FUNCTION_BLOCK FB_CHPSystem EXTENDS FB_SystemContinous
VAR_INPUT
	aHeatCounterTelegramm : ARRAY[1..cMBUS_MaxTelegrams] OF ST_MBus_Data2;
END_VAR
VAR_OUTPUT
	bSetStatusOnFeedback : BOOL; //Feedback if CHP unit should be switched on to be sent to supply air valve
END_VAR
VAR	
	//chp
	CHP : FB_CHP;

	//pump
	stPU32xDefaultParameters : ST_PumpGrundfosMagna3DefaultParameters;
	PU32x : FB_PumpGrundfosMagna3 := (ST_DefaultParameters := stPU32xDefaultParameters);
	
	//valves
	stSV32xDefaultParameters : ST_DiscreteValveDefaultParameters := (nFeedback := 3);
	stRV32xDefaultParameters : ST_MixingValveDefaultParameters := (bFeedbackSignal := TRUE, tTaskCycleTime := GlobalVariables.tTaskCycleTime_MAIN, tCtrlCycleTime := GlobalVariables.tCtrlCycleTime_MAIN);	
	SV32x : FB_DiscreteValve := (ST_DefaultParameters := stSV32xDefaultParameters);
	RV32x : FB_MixingValve := (ST_DefaultParameters := stRV32xDefaultParameters);
	WMZ32x : FB_MollineC3HeatCounter();
	
	//internal variables
	bSetStatusOn_CHP   : BOOL;
	bSetStatusOn_PU32x : BOOL;
	bSetStatusOn_SV32x : BOOL;
	bSetStatusOn_RV32x : BOOL; 	
	
	//timer
	bStartTimer : BOOL;
	Timer : TON;
END_VAR

bSetStatusOnFeedback := bSetStatusOn;

//use timer because valve has no feedback signal (75 sec)
Timer(IN := bStartTimer,
	PT := T#75S);

MAIN();
CHP.GetState();
CHP(fSetPointAutomatic := 100,
	bSetStatusOnAutomatic := bSetStatusOn_CHP,
	bAlgorithmPermission := bAlgorithmPermission,
	nControlModeAutomatic := 0,
	fExternalFeedTemperature := PU32x.fTemperatureInternal);
CHP.SetState();

SV32x.GetState_BI();
SV32x(bSetStatusOnAutomatic := bSetStatusOn_SV32x,
	bAlgorithmPermission := bAlgorithmPermission);
SV32x.SetState_BO();

RV32x.GetState_AI();
RV32x(fSetPointAutomatic := fSetPoint,
	bSetStatusOnAutomatic := bSetStatusOn_RV32x,
	bAlgorithmPermission := bAlgorithmPermission,
	fTemperatureExternal := PU32x.fTemperatureInternal,
	nControlModeAutomatic := 2);
RV32x.SetState_AO();

PU32x.GetState_Profibus();
PU32x(fSetPointAutomatic := 100,
	bSetStatusOnAutomatic := bSetStatusOn_PU32x,
	bAlgorithmPermission := bAlgorithmPermission,
	nControlModeAutomatic := 0);
PU32x.SetState_Profibus();

WMZ32x(aHeatCounterTelegramm := aHeatCounterTelegramm);

METHOD PROTECTED  CheckError : BOOL
VAR_INPUT
END_VAR
VAR
	bError_PU32x : BOOL;
	//bError_CHP : BOOL;
END_VAR
VAR_OUTPUT
	bError : BOOL;
END_VAR
//check pumps for errors
bError_PU32x := PU32x.bError;
//bError_CHP := CHP.bError;

//bError := bError_PU32x OR bError_CHP;
bError := bError_PU32x;
END_METHOD

METHOD PROTECTED  Operational : BOOL
VAR_INPUT
END_VAR
VAR_OUTPUT
	bSwitchToWorking : BOOL := FALSE;
END_VAR
bSetStatusOn_CHP := TRUE;

//IF CHP.bStatusOn THEN
bStartTimer := TRUE;
IF TIMER.Q THEN
	bSwitchToWorking := TRUE;
	bStartTimer := FALSE;
END_IF
END_METHOD

METHOD PROTECTED  RampDown : BOOL
VAR_INPUT
END_VAR
VAR_OUTPUT
	bRampDownFinished : BOOL := FALSE;
END_VAR
bSetStatusOn_CHP := FALSE;

//IF NOT CHP.bStatusOn THEN
bStartTimer := TRUE;
IF Timer.Q THEN
	bSetStatusOn_PU32x := FALSE;
	bStartTimer := FALSE;
END_IF

IF NOT PU32x.bStatusOn THEN
	bSetStatusOn_RV32x := FALSE;
	bSetStatusOn_SV32x := FALSE;

	IF SV32x.bStatusOn THEN
		bRampDownFinished := TRUE;
	END_IF
END_IF
END_METHOD

METHOD PROTECTED  RampUp : BOOL
VAR_INPUT
END_VAR
VAR_OUTPUT
	bRampUpFinished : BOOL := FALSE;
END_VAR
bSetStatusOn_SV32x := TRUE;
bSetStatusOn_RV32x := TRUE;

IF SV32x.bStatusOn THEN
	bSetStatusOn_PU32x := TRUE;
END_IF

IF PU32x.bStatusOn THEN
	bStartTimer := FALSE; //resets timer	
	bRampUpFinished := TRUE;
END_IF
END_METHOD

METHOD PROTECTED   SetSetPointLimits : BOOL
VAR_INPUT
END_VAR
aSetPointLimits[1] := CHP.ST_DefaultParameters.aSetPointLimitsTemperature[1];
aSetPointLimits[2] := CHP.ST_DefaultParameters.aSetPointLimitsTemperature[2];
END_METHOD

METHOD PROTECTED  Working : BOOL
VAR_INPUT
END_VAR
VAR_OUTPUT
	bSwitchToOperational : BOOL := FALSE;
END_VAR
//empty method
END_METHOD

END_FUNCTION_BLOCK

(* stored: Version 1.1.0.1, ProductVersion 3.1.4024.10
   POU FB_CHPSystem: Id {03be9f87-4e59-4877-a478-dceefb67f1c9}, SpecialFunc None
   Method CheckError: Id {684c4c5f-5b63-4ac1-a5ee-1759d03ff526}
   Method Operational: Id {1a1d7ebc-5ebc-49ca-9755-166e1ea8616e}
   Method RampDown: Id {0de23c98-c56a-469e-955b-2ff61016c0ab}
   Method RampUp: Id {3071767d-8111-44da-af02-b65d0afaa40d}
   Method SetSetPointLimits: Id {8cfe0602-4afb-47e7-b900-5c78610daffb}
   Method Working: Id {6321a476-f7aa-4875-ae31-cebd1b5c7895} *)
